(* Logix 5000 project; controller Ex_2_07 Emulate 5570 rev 33.11; software revision 33.00 *)
// Turn on lamp with two push buttons (NO,NC)

TASK MainTask (continuous, watchdog 500 ms) : MainProgram

MODULES
   Local : Emulate 5570 (ICP 4, rev 33.11)
END_MODULES

VAR_GLOBAL   (* controller tags *)
   P1 : BOOL;   // Lamp P1
   S1 : BOOL;   // Push Button S1
   S2 : BOOL;   // Push Button S2
END_VAR

PROGRAM MainProgram   (* main routine MainRoutine *)

ROUTINE MainRoutine   (* ladder *)
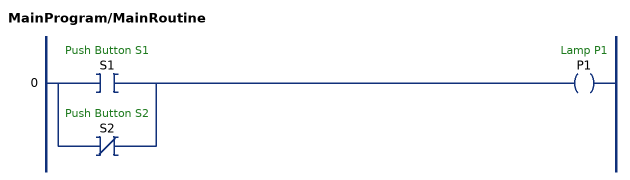
   0: [XIC(S1) ,XIO(S2) ]OTE(P1);
END_ROUTINE
END_PROGRAM
